# EPICS autosave request: iocBoot/lakeshoreCommon.req
$(P):DESC1
$(P):DESC2
$(P):DESC3
$(P):DESC4
$(P):readAll.SCAN
